(* IEC 61131-3 sources: SIGMATEK-Jumag-Utils-Examples/twoPointController/Class/Class0, 1 file *)

(* ---- Class0.st ---- *)
(*!
<Class
	Name               = "Class0"
	Revision           = "0.0"
	RealtimeTask       = "false"
	CyclicTask         = "true"
	DefCyclictime      = "10 ms"
	BackgroundTask     = "false"
	Sigmatek           = "false"
	OSInterface        = "false"
	HighPriority       = "false"
	Automatic          = "false"
	UpdateMode         = "Prescan"
	SharedCommandTable = "true"
	Objectsize         = "(540,240)">
	<Channels>
		<Server Name="ClassSvr" Visualized="false" Initialize="false" WriteProtected="true" Retentive="false"/>
		<Server Name="Off_Setpoint" Visualized="false" Initialize="true" WriteProtected="false" Retentive="false"/>
		<Server Name="On_Setpoint" Visualized="false" Initialize="true" WriteProtected="false" Retentive="false"/>
		<Client Name="SignalGenerator" Required="true" Internal="false"/>
	</Channels>
	<Dependencies>
		<Files>
			<File Path=".\Source\controller.c"/>
		</Files>
	</Dependencies>
</Class>
*)
Class0 : CLASS
  //Servers:
	ClassSvr 	: SvrChCmd_DINT;
	On_Setpoint 	: SvrCh_DINT;
	Off_Setpoint 	: SvrCh_DINT;
  //Clients:
	SignalGenerator 	: CltCh_DINT;
  //Variables:
		oldState 	: BOOL;
  //Functions:

	FUNCTION VIRTUAL GLOBAL CyWork
		VAR_INPUT
			EAX 	: UDINT;
		END_VAR
		VAR_OUTPUT
			state (EAX) 	: UDINT;
		END_VAR;
  //Tables:
	FUNCTION @STD
		VAR_OUTPUT
			ret_code	: CONFSTATES;
		END_VAR;
	FUNCTION GLOBAL TAB @CT_;
END_CLASS;

Function Global __cdecl twoPointCtrl
VAR_INPUT
  INPUT : DINT;
  ON_Setpoint : DINT;
  OFF_Setpoint : DINT;
  pOld : ^BOOL;
END_VAR
VAR_OUTPUT
  Q : BOOL;
END_VAR;

FUNCTION VIRTUAL GLOBAL Class0::CyWork
	VAR_INPUT
		EAX 	: UDINT;
	END_VAR
	VAR_OUTPUT
		state (EAX) 	: UDINT;
	END_VAR

  SignalGenerator := SignalGenerator.Read();

  ClassSvr := twoPointCtrl( INPUT := SignalGenerator,
                            ON_Setpoint:= On_Setpoint,
                            OFF_Setpoint:= Off_Setpoint,
                            pOld:= #oldState);

	state := READY;

END_FUNCTION
